// TIA Portal project "Açık Kapalı Kontak Uygulaması" (V18)

(* hardware
DEVICE "S7-1200 station_1"  S7-1200 Station
   slot 0: "Rack_0"  S7-1200 Rack  Rack  V1.0
   slot 1: "PLC_1"  CPU 1214C AC/DC/Rly  6ES7 214-1BG40-0XB0  V4.6
*)

// ===== PLC "PLC_1"  CPU 1214C AC/DC/Rly =====

VAR_GLOBAL   // PLC tag table "Default tag table"
   "Stop" AT %I0.0 : Bool;
   "Start_1" AT %I0.1 : Bool;
   "Start_2" AT %I0.2 : Bool;
   "Motor_1" AT %Q0.0 : Bool;
   "Start_3" AT %I0.3 : Bool;
   "Motor_2" AT %Q0.1 : Bool;
   "Motor_3" AT %Q0.2 : Bool;
END_VAR

ORGANIZATION_BLOCK "Main"   // OB1, LAD, ProgramCycle
TITLE = "Main Program Sweep (Cycle)"
{ S7_Optimized_Access := 'TRUE' }
VERSION : 0.1
   VAR_INPUT
      Initial_Call : Bool;   // Initial call of this OB
      Remanence : Bool;   // =True, if remanent data are available
   END_VAR
BEGIN

REGION Network 1
   // Maksimum 3 girişin olduğu bir sistemde çıkış şu şartlara bağlı olacaktır.
   //            2 giriş olduğunda Q0.0 aktif olacak.
   //            3 giriş olduğunda Q0.1 aktif olacak.
   //            1 giriş aktif iken ise Q0.2 aktif olacaktır.
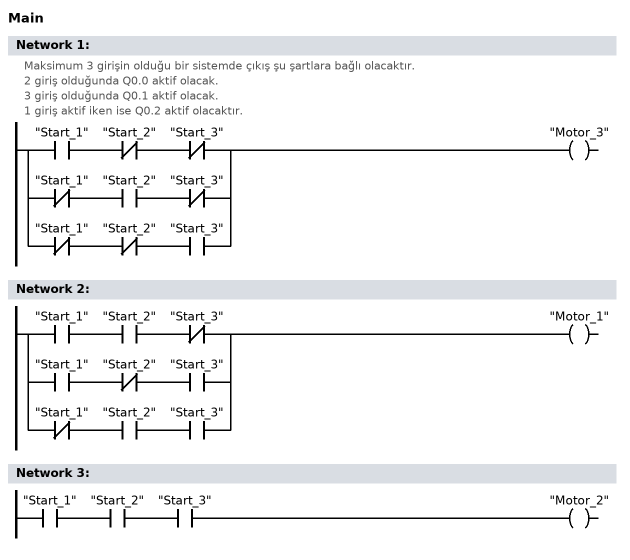
   RUNG wire#powerrail
      Contact( "Start_1" )
      I_Contact( "Start_2" )
      I_Contact( "Start_3" )
      wire#w1
      Coil( "Motor_3" )
   END_RUNG
   RUNG wire#powerrail
      I_Contact( "Start_1" )
      Contact( "Start_2" )
      I_Contact( "Start_3" )
   END_RUNG wire#w1
   RUNG wire#powerrail
      I_Contact( "Start_1" )
      I_Contact( "Start_2" )
      Contact( "Start_3" )
   END_RUNG wire#w1
   // the same network as SCL:
   "Motor_3" := ("Start_1" AND NOT "Start_2" AND NOT "Start_3") OR (NOT "Start_1" AND "Start_2" AND NOT "Start_3") OR (NOT "Start_1" AND NOT "Start_2" AND "Start_3");
END_REGION

REGION Network 2
   RUNG wire#powerrail
      Contact( "Start_1" )
      Contact( "Start_2" )
      I_Contact( "Start_3" )
      wire#w1
      Coil( "Motor_1" )
   END_RUNG
   RUNG wire#powerrail
      Contact( "Start_1" )
      I_Contact( "Start_2" )
      Contact( "Start_3" )
   END_RUNG wire#w1
   RUNG wire#powerrail
      I_Contact( "Start_1" )
      Contact( "Start_2" )
      Contact( "Start_3" )
   END_RUNG wire#w1
   // the same network as SCL:
   "Motor_1" := ("Start_1" AND "Start_2" AND NOT "Start_3") OR ("Start_1" AND NOT "Start_2" AND "Start_3") OR (NOT "Start_1" AND "Start_2" AND "Start_3");
END_REGION

REGION Network 3
   RUNG wire#powerrail
      Contact( "Start_1" )
      Contact( "Start_2" )
      Contact( "Start_3" )
      Coil( "Motor_2" )
   END_RUNG
   RUNG wire#powerrail
   END_RUNG
   // the same network as SCL:
   "Motor_2" := "Start_1" AND "Start_2" AND "Start_3";
END_REGION
END_ORGANIZATION_BLOCK